INTERFACE ITF_Track

PROPERTY Length : LREAL
GET
END_GET
SET
END_SET
END_PROPERTY

END_INTERFACE

(* stored: Version 1.1.0.1, ProductVersion 3.1.4024.12
   Itf ITF_Track: Id {0d5dfb01-5a03-4dd3-bd30-13a53a2b2ab7}
   Property Length: Id {13472377-55c8-49d9-a155-542f2fe93014}
   Get Get: Id {1c8c8e06-3b55-4c8e-9316-70024955f4a4}
   Set Set: Id {575fe15a-a4b8-49f8-848f-c7116dcfdcc8} *)
